FUNCTION_BLOCK FB_VISU_VAC_VALVE 
VAR_INPUT
END_VAR
VAR_OUTPUT
END_VAR
VAR
	itfVacValve: I_VAC_VALVE;
	itfOpMode: I_OP_MODE;
	strFullObjectName: STRING;
	strInfo: STRING;
	bVacOn: BOOL;
	bBlowOn: BOOL;
	bBlowOrVac: BOOL;   
	bVakOk: BOOL; 
	bActivateVac: BOOL;
	bActivateBlow: BOOL;   
	bActivateOff: BOOL;  
	bFrameInvisible: BOOL:= TRUE;
	stEvent: ST_EVENT;                                                                                                                      
END_VAR

IF NOT (itfOpMode.P_OP_MODE_STATE= OP_MODE.MANUAL) THEN
	bFrameInvisible:=TRUE;
END_IF

IF itfVacValve.P_STATE= E_PNEU_VAC_VALVE.AllOff THEN
	strInfo:= F_RET_TXTLIST_ENTRY(strPortNr:= '851', strID:='14', strTxtLstName:= 'TXT_LIST_PNEMATIC_ACTOR');
	bVacOn:=FALSE;
	bBlowOn:=FALSE;
	bVakOk:=FALSE;	
END_IF

IF itfVacValve.P_STATE= E_PNEU_VAC_VALVE.Blowing THEN
	strInfo:= F_RET_TXTLIST_ENTRY(strPortNr:= '851', strID:='13', strTxtLstName:= 'TXT_LIST_PNEMATIC_ACTOR');
	bVacOn:=FALSE;
	bBlowOn:=TRUE;	
	bVakOk:=FALSE;
END_IF

IF itfVacValve.P_STATE= E_PNEU_VAC_VALVE.Vac_ON_NotDetect THEN
	strInfo:= F_RET_TXTLIST_ENTRY(strPortNr:= '851', strID:='11', strTxtLstName:= 'TXT_LIST_PNEMATIC_ACTOR');
	bVacOn:=TRUE;
	bBlowOn:=FALSE;	
	bVakOk:=FALSE;
END_IF

IF itfVacValve.P_STATE= E_PNEU_VAC_VALVE.VacDetect THEN
	strInfo:= F_RET_TXTLIST_ENTRY(strPortNr:= '851', strID:='12', strTxtLstName:= 'TXT_LIST_PNEMATIC_ACTOR');
	bVacOn:=TRUE;
	bBlowOn:=FALSE;	
	bVakOk:=TRUE;
END_IF

strFullObjectName:= itfVacValve.P_FullObjectPath;
bBlowOrVac:=bVacOn OR bBlowOn;

IF (itfOpMode.P_OP_MODE_STATE=OP_MODE.MANUAL) THEN
	IF bActivateVac THEN
		itfVacValve.M_Vac();
	END_IF
	IF bActivateBlow THEN
		itfVacValve.M_Blow();
	END_IF
	IF bActivateOff THEN
		itfVacValve.M_AllOff();
	END_IF
ELSE
	bActivateVac:=FALSE;
	bActivateBlow:= FALSE;
	bActivateOff:= FALSE;
END_IF

stEvent:= itfVacValve.P_Event;

METHOD FB_init : BOOL
VAR_INPUT
	bInitRetains : BOOL; // if TRUE, the retain variables are initialized (warm start / cold start)
	bInCopyCode : BOOL;  // if TRUE, the instance afterwards gets moved into the copy code (online change)
	itfVacValve: I_VAC_VALVE;
	itfOpMode: I_OP_MODE;
END_VAR
THIS^.itfVacValve:= itfVacValve;
THIS^.itfOpMode:= itfOpMode;
END_METHOD

END_FUNCTION_BLOCK

(* stored: Version 1.1.0.1, ProductVersion 3.1.4024.12
   POU FB_VISU_VAC_VALVE: Id {8c62bd0b-96f6-4f37-a5b2-bacd54a8806f}, SpecialFunc None
   Method FB_init: Id {682b31ce-f8d2-4d55-918e-ce2c1024dcab} *)
